(* IEC 61131-3 sources: std_i2980_v2.06_cp053/Source/IMM/ieccontrol/ODC1 (part 11) *)

IF sv_DataState = nReadMoldData THEN
   //loading of mold data in progress
   mbIgnoreProgramSwitchChange := TRUE;
   PrevState := nReadMoldData;
   sv_SequenceDimension.iMaxColumns := 0;
   sv_SequenceDimension.iMaxRows := 0;
ELSIF sv_DataState = nReadSequenceData THEN
   //loading of sequence in progress
   mbIgnoreProgramSwitchChange := TRUE;
   PrevState := nReadSequenceData;
   sv_SequenceDimension.iMaxColumns := 0;
   sv_SequenceDimension.iMaxRows := 0;
END_IF;

IF sv_DataState = nReady AND mbIgnoreProgramSwitchChange THEN

   //loading procedure ready
   mbIgnoreProgramSwitchChange := FALSE;

   //decide if only conditions should be recalculated (after loading sequence)
   //or complete sequence should be created (after program switch changed)
   IF sv_bUseProgramSwitches THEN
      aSetPendingRecalc(RecalcMode := nODCRecalcReloadFiles);
   ELSIF PrevState = nReadMoldData THEN
      aSetPendingRecalc(RecalcMode := nODCRecalcInternal);
   ELSIF PrevState = nReadSequenceData THEN
      aSetPendingRecalc(RecalcMode := nODCRecalcInternal);
   END_IF;

   aDoPendingRecalc();
   IF aDoPendingRecalc.bStartedRecalc THEN
      fbDebugTrace2(nDeviceState, 'recalc because data state change');
   END_IF;

   PrevState := nReady;
END_IF;

@END_Body

@@@BEG_Comment@@@
@TL(0)

@@@END_Comment@@@

@BEG_Body
@TL(34)
(**************************************** WARNING ********************************************
 *** The KEBA Kemro K2 System including software is not intended for safety control tasks! ***
 ***                       For further information see Comment tab!                        ***
 *********************************************************************************************)

IF NOT sv_bODCFilesChanged THEN
   RETURN;
END_IF;

sv_bODCFilesChanged := FALSE;

IF NOT sv_bInitDone THEN
   fbDebugTrace('ignoring sv_bODCFilesChanged because sv_bInitDone is FALSE');
   RETURN;
END_IF;

(* rebuild ODC array immediately with reloading files *)
aSetPendingRecalc(RecalcMode := nODCRecalcReloadFiles);

IF sv_OperationMode >= nHalfAutomatic THEN
   fbDebugTrace('skipping ODC recalc after file change because of OperationMode');
   RETURN;
END_IF;

IF sv_StartedMovements.iStartedMovements > 0 THEN
   fbDebugTrace('skipping ODC recalc after file change because there are started movements');
   RETURN;
END_IF;

aDoPendingRecalc();
IF aDoPendingRecalc.bStartedRecalc THEN
   fbDebugTrace2(nDeviceState, 'recalc because files changed');
END_IF;

@END_Body

@@@BEG_Comment@@@
@TL(1)
React to program switch changes, and recalculate the ODC sequence.
@@@END_Comment@@@

@BEG_Body
@TL(38)
(**************************************** WARNING ********************************************
 *** The KEBA Kemro K2 System including software is not intended for safety control tasks! ***
 ***                       For further information see Comment tab!                        ***
 *********************************************************************************************)

IF sv_iActiveEditors <> 0 THEN
   //teach mode active
   //avoid changing operation mode to HA or FA
   fbLockUnlock.Alarm.AlarmId := erTeachModeActive;
   fbLockUnlock.Mode := nLockAbort;
   fbLockUnlock();

   //reset sv_bUseProgramSwitches immediately after activating teach mode
   //so that "controlled by machine sequencer" is displayed instead of program switches
   sv_bUseProgramSwitches := FALSE;
   RETURN;
ELSE
   fbLockUnlock.Alarm.AlarmId := erTeachModeActive;
   fbLockUnlock.Mode := nUnlock;
   fbLockUnlock();
END_IF;

//teach mode inactive => new sequence programmed by editor
// -> create internal array, calculate safety conditions, do plaus checks
aSetPendingRecalc(RecalcMode := nODCRecalcInternal);

aDoPendingRecalc();
IF aDoPendingRecalc.bStartedRecalc THEN
   fbDebugTrace2(nDeviceState, 'recalc because new sequence from editor');
END_IF;

@END_Body

@@@BEG_Comment@@@
@TL(2)
create internal array and calculate safety conditions after
teachmode becomes inactive
@@@END_Comment@@@

@BEG_Body
@TL(25)
(**************************************** WARNING ********************************************
 *** The KEBA Kemro K2 System including software is not intended for safety control tasks! ***
 ***                       For further information see Comment tab!                        ***
 *********************************************************************************************)

IF sv_iSequenceToRestore = 0 THEN
   RETURN;
END_IF;

IF sv_iSequenceToRestore > cODCSequenceBackupCount THEN
   fbDebugTrace2(nODCInterpreter, 'restoring actual sequence calculated from switches');
   aSetPendingRecalc(RecalcMode := nODCRecalcCylce);
END_IF;

fbDebugTrace2(nODCInterpreter, CONCAT('restoring old sequence ', DINT_TO_STRING(sv_iSequenceToRestore)));
sv_ODCSequence := sv_ODCSequenceBackup[sv_iSequenceToRestore].Sequence;
aSetPendingRecalc(RecalcMode := nODCRecalcSafety);
aDoPendingRecalc(); //FIXME: this may not do more than security recalculation -> otherwise loaded array would be overwritten
IF aDoPendingRecalc.bStartedRecalc THEN
   fbDebugTrace2(nDeviceState, 'recalc because sequence backup is restored');
END_IF;
sv_iSequenceToRestore := 0;
fbDebugTrace2(nODCInterpreter, 'restoring old sequence done');

@END_Body

@@@BEG_Comment@@@
@TL(0)

@@@END_Comment@@@

@BEG_Body
@TL(45)
(**************************************** WARNING ********************************************
 *** The KEBA Kemro K2 System including software is not intended for safety control tasks! ***
 ***                       For further information see Comment tab!                        ***
 *********************************************************************************************)

IF NOT sv_bProgramSwitchChanged THEN
   RETURN;
END_IF;

sv_bProgramSwitchChanged := FALSE;

IF NOT sv_bInitDone THEN
   fbDebugTrace2(nODCInterpreter, 'ignoring program switch change because sv_bInitDone is FALSE');
   RETURN;
END_IF;

IF NOT sv_bUseProgramSwitches THEN
   // ignore changing of program switch if sequence from graphical editor is used
   fbDebugTrace2(nODCInterpreter, 'ignoring program switch change because of sv_bUseProgramSwitches');
   RETURN;
END_IF;

IF mbIgnoreProgramSwitchChange THEN
   fbDebugTrace2(nODCInterpreter, 'ignoring program switch change because of sv_DataState');
   RETURN;
END_IF;

aSetPendingRecalc(RecalcMode := nODCRecalcCylce);

IF sv_OperationMode >= nHalfAutomatic THEN
   fbDebugTrace('skipping ODC recalc after program switch change because of OperationMode');
   RETURN;
END_IF;

IF sv_StartedMovements.iStartedMovements > 0 THEN
   fbDebugTrace('skipping ODC recalc after program switch change because there are started movements');
   RETURN;
END_IF;

(* rebuild ODC array immediately without reloading files *)
aDoPendingRecalc();
IF aDoPendingRecalc.bStartedRecalc THEN
   fbDebugTrace2(nDeviceState, 'recalc because program switch changed');
END_IF;

@END_Body

@@@BEG_Comment@@@
@TL(1)
React to program switch changes, and recalculate the ODC sequence.
@@@END_Comment@@@

@BEG_Body
@TL(39)
(**************************************** WARNING ********************************************
 *** The KEBA Kemro K2 System including software is not intended for safety control tasks! ***
 ***                       For further information see Comment tab!                        ***
 *********************************************************************************************)

IF NOT sv_bActivationChanged THEN
   RETURN;
END_IF;

sv_bActivationChanged := FALSE;

IF NOT sv_bInitDone THEN
   fbDebugTrace('ignoring sv_bActivationChanged because sv_bInitDone is FALSE');
   RETURN;
END_IF;

IF mbIgnoreProgramSwitchChange THEN
   fbDebugTrace2(nODCInterpreter, 'ignoring activation change because of sv_DataState');
   RETURN;
END_IF;

(* recalculate ODC safety without reloading files/recalculating the sequence *)
aSetPendingRecalc(RecalcMode := nODCRecalcSafety);

IF sv_OperationMode >= nHalfAutomatic THEN
   fbDebugTrace('skipping ODC recalc after activation change because of OperationMode');
   RETURN;
END_IF;

IF sv_StartedMovements.iStartedMovements > 0 THEN
   fbDebugTrace('skipping ODC recalc after activation change because there are started movements');
   RETURN;
END_IF;

aDoPendingRecalc();
IF aDoPendingRecalc.bStartedRecalc THEN
   fbDebugTrace2(nDeviceState, 'recalc because activation change');
END_IF;

@END_Body

@@@BEG_Comment@@@
@TL(1)
React to program switch changes, and recalculate the ODC sequence.
@@@END_Comment@@@

@BEG_Body
@TL(8)
(**************************************** WARNING ********************************************
 *** The KEBA Kemro K2 System including software is not intended for safety control tasks! ***
 ***                       For further information see Comment tab!                        ***
 *********************************************************************************************)

b := FCreateODCVersion();
STOP_PROCESS_ALGORITHM();

@END_Body

@@@BEG_Comment@@@
@TL(0)

@@@END_Comment@@@

@BEG_Body
@TL(29)
(**************************************** WARNING ********************************************
 *** The KEBA Kemro K2 System including software is not intended for safety control tasks! ***
 ***                       For further information see Comment tab!                        ***
 *********************************************************************************************)

IF mbIgnoreProgramSwitchChange THEN
   //loading procedure in progress
   RETURN;
END_IF;

IF sv_bUseProgramSwitches THEN
   //activate all devices after a change from
   //machine sequencer mode to program switch mode
   FOR iDevice := 1 TO sv_ODCDeviceMovements.iCount DO
      IF CHECK_REF(sv_ODCDeviceMovements.Devices[iDevice].pbDeviceActivated^) THEN
         sv_ODCDeviceMovements.Devices[iDevice].pbDeviceActivated^ := TRUE;
      END_IF;
   END_FOR;

   //create new sequence depending on the program switches
   //set mode to nODCRecalcReloadFiles because maybe sequence was
   //never created with program switches before
   aSetPendingRecalc(RecalcMode := nODCRecalcReloadFiles);
   aDoPendingRecalc();
   IF aDoPendingRecalc.bStartedRecalc THEN
      fbDebugTrace2(nDeviceState, 'recalc because change to program switch mode');
   END_IF;
END_IF;

@END_Body

@@@BEG_Comment@@@
@TL(1)
trigger creation of sequence by program switches
@@@END_Comment@@@

@BEG_Body
@TL(78)
(**************************************** WARNING ********************************************
 *** The KEBA Kemro K2 System including software is not intended for safety control tasks! ***
 ***                       For further information see Comment tab!                        ***
 *********************************************************************************************)

Pos.iColumn := 1;
Pos.iRow := 1;

DeviceId.CompId := sv_ODCSequence[1,1].iCompId;
DeviceId.IndexId := INT_TO_DINT(sv_ODCSequence[1,1].iIndexId);

//check safety array of first step (ODC.BeginSequence)
bEjectorIgnored := FALSE;
IF mbEjeBwdAtCycleStart THEN
   //ejector must not be bwd when operator switches to HA or FA
   //the ejector bwd movement is done in aRunAutoCylce
   //=> start of cycle should be possible if ejector is not bwd)
   //=> dependency must be modified for this case
   //all other safety relevant movements (mold, cores, ...) must be in the calculated startposition
   EjectorDependency := sv_ODCSequenceInt[1,1].SafetyArray[miIndexEjectorInSafetyArray].Dependency;
   sv_ODCSequenceInt[1,1].SafetyArray[miIndexEjectorInSafetyArray].Dependency := cNoDependency;
   bEjectorIgnored := TRUE;
END_IF;

//check init safety array
//(check all safety relevant devices)
abODCCheckDependencies.aCheck(StepPos := Pos, DeviceIdSelf := DeviceId);
bAllowed := abODCCheckDependencies.aCheck.bAllowed;

//write back the original value
IF bEjectorIgnored THEN
   sv_ODCSequenceInt[1,1].SafetyArray[miIndexEjectorInSafetyArray].Dependency := EjectorDependency;
END_IF;

//check state of not safety relevant devices
//always check even if safety relevant check already failed
SafetyArray := sv_ODCSequenceInt[1,1].SafetyArray;
FOR iDevice := 1 TO sv_ODCDeviceMovements.iCount DO
   DeviceId := sv_ODCDeviceMovements.Devices[iDevice].DeviceId;
   iDefaultMove := sv_ODCDeviceMovements.Devices[iDevice].iDefaultMoveNumber;

   IF (SafetyArray[iDevice].Dependency = cNoDependency) AND (DeviceId.CompId <> cCompODC) THEN
      //device not safety relevant
      IF sv_ODCDeviceMovements.Devices[iDevice].pbDeviceActivated^ AND iDefaultMove <> 0 THEN
         //if device is activated and a default movement is available,
         //the default movement of this device must be in endposition
         fbCheckPosReached(DeviceId := DeviceId,
                           MoveDir := sv_MovementsAvailable[iDefaultMove].pMovementData^.MoveDir,
                           MoveId := sv_MovementsAvailable[iDefaultMove].pMovementData^.MoveId);

         IF NOT fbCheckPosReached.bPosReached THEN
            IF sv_TraceLevel.bODCInterpreter THEN
               fbDebugTrace(CONCAT('cycle start not allowed by default position check of ',
                                   DINT_TO_STRING(DeviceId.CompId), '.', DINT_TO_STRING(DeviceId.IndexId),
                                   ' -> setting alarm ',
                                   GET_ALARM_NAME(fbCheckPosReached.Alarm.AlarmId)));
            END_IF;
            //set according alarm
            SET_ALARM(Name := fbCheckPosReached.Alarm.AlarmId,
                      SubID1 := fbCheckPosReached.Alarm.SubId[1],
                      SubID2 := fbCheckPosReached.Alarm.SubId[2],
                      SubID3 := fbCheckPosReached.Alarm.SubId[3],
                      SubID4 := fbCheckPosReached.Alarm.SubId[4]);
            bAllowed := FALSE;
         END_IF;
      END_IF;
   END_IF;
END_FOR;

IF NOT bAllowed THEN
   IF sv_TraceLevel.bODCInterpreter THEN
      fbDebugTrace('checking cycle start conditions found problems -> switching back to manual mode');
   END_IF;
   //switch away from auto mode if any check fails
   fbAutoManual();
END_IF;

@END_Body

@@@BEG_Comment@@@
@TL(6)
This algorithm checks the start conditions for the cycle if the
operator switches to half or fullauto cycle.
Safety relevant devices must be in the position which they should have according
the programmed cycle.
Not safety relevant devices must be in their default position.
Deactivated devices and devices which have no default position are not checked.
@@@END_Comment@@@

@BEG_Body
@TL(28)
(**************************************** WARNING ********************************************
 *** The KEBA Kemro K2 System including software is not intended for safety control tasks! ***
 ***                       For further information see Comment tab!                        ***
 *********************************************************************************************)

IF sv_TraceLevel.bODCInterpreter THEN
   //trace opmode switch
   IF sv_OperationMode = nSetup THEN
      sOperationMode := 'Setup';
   ELSIF sv_OperationMode = nManual THEN
      sOperationMode := 'Manual';
   ELSIF sv_OperationMode = nHalfAutomatic THEN
      sOperationMode := 'HalfAutomatic';
   ELSIF sv_OperationMode = nFullAutomatic THEN
      sOperationMode := 'FullAutomatic';
   ELSE
      sOperationMode := '???';
   END_IF;
   fbDebugTrace(CONCAT('sv_OperationMode changed to ', sOperationMode));
END_IF;

IF PrevOpMode < nHalfAutomatic AND sv_OperationMode >= nHalfAutomatic THEN
   //check cycle start conditions
   aCheckCycleStartConditions();
END_IF;

PrevOpMode := sv_OperationMode;

@END_Body

@@@BEG_Comment@@@
@TL(0)

@@@END_Comment@@@

@BEG_SfcBody
25 16 17

@BEG_SfcData 2
@StepSeq @RT(4)sseq @F 3
@Step @RT(5)SInit @F @T @F @F @RT(0) @F
@AcbCont @RT(7)unnamed @F 0

@Trans @RT(6)Trans1 @F @T @F @F @T @F @TL(2)
TRUE

@RT(6)Trans1 @F
@Loop @RT(4)loop @F 2
@StepSeq @RT(3)seq @F 5
@Step @RT(5)S_Run @F @F @F @F @RT(0) @F
@AcbCont @RT(7)unnamed @F 2
@Acb @RT(8)Action24 @F @T @RT(1)P @RT(0) @F @F @T @TL(2)
sv_bODCCombinedMoveActive := TRUE;

@F
@Acb @RT(20)ARunCombinedMovement @F @T @RT(1)N @RT(0) @F @F @T @TL(4)
// run a combined movements
abInterpreter.aInterpret();
abInterpreter.aStatus();

@F

@AltBranch @RT(3)alt @F 3
@TransSeq @RT(4)tseq @F 5
@Trans @RT(9)TFinished @F @T @F @F @T @F @TL(2)
abInterpreter.aStatus.bFinished

@RT(6)Trans2 @F
@Step @RT(10)S_Finished @F @F @F @F @RT(0) @F
@AcbCont @RT(7)unnamed @F 1
@Acb @RT(6)ATrace @F @F @RT(1)P @RT(0) @F @F @F @F

@Trans @RT(18)TAllMovementsReady @F @T @F @F @T @F @TL(2)
sv_StartedManualMovements.iStartedMovements = 0

@RT(6)Trans7 @T @TL(2)
Interpreter is finished -> wait untill all movements
are ready  (for example airvalve can still be active)

@Step @RT(17)S_StopInterpreter @F @F @F @F @RT(0) @F
@AcbCont @RT(7)unnamed @F 1
@Acb @RT(16)AStopInterpreter @F @T @RT(1)P @RT(0) @F @F @T @TL(2)
abInterpreter.aStopInterpreterNormal();

@F

@Trans @RT(7)Trans11 @F @T @F @F @T @F @TL(2)
TRUE

@RT(7)Trans11 @F

@TransSeq @RT(4)tseq @F 3
@Trans @RT(10)TNotActive @F @T @F @F @T @F @TL(2)
NOT abInterpreter.aStatus.bActive

@RT(6)Trans5 @F
@Step @RT(11)S_NotActive @F @F @F @F @RT(0) @F
@AcbCont @RT(7)unnamed @F 1
@Acb @RT(15)ATraceNotActive @F @F @RT(1)P @RT(0) @F @F @F @F

@Trans @RT(6)Trans8 @F @T @F @F @T @F @TL(2)
TRUE

@RT(6)Trans8 @F

@TransSeq @RT(4)tseq @F 3
@Trans @RT(6)TError @F @T @F @F @T @F @TL(2)
abInterpreter.aStatus.bError

@RT(6)Trans6 @F
@Step @RT(7)S_Error @F @F @F @F @RT(0) @F
@AcbCont @RT(7)unnamed @F 1
@Acb @RT(11)ATraceError @F @F @RT(1)P @RT(0) @F @F @F @F

@Trans @RT(6)Trans9 @F @T @F @F @T @F @TL(2)
TRUE

@RT(6)Trans9 @F

@Step @RT(8)S_Recalc @F @F @F @F @RT(0) @F
@AcbCont @RT(7)unnamed @F 1
@Acb @RT(16)ADoPendingRecalc @F @F @RT(1)P @RT(0) @F @F @F @F

@Trans @RT(7)Trans12 @F @T @F @F @T @F @TL(2)
TRUE

@RT(7)Trans12 @F
@Step @RT(6)S_Stop @F @F @F @F @RT(0) @F
@AcbCont @RT(7)unnamed @F 1
@Acb @RT(5)AStop @F @T @RT(1)P @RT(0) @F @F @T @TL(3)
sv_bODCCombinedMoveActive := FALSE;
STOP_PROCESS_ALGORITHM();

@F

@Trans @RT(6)Trans4 @F @T @T @T @T @T @TL(2)
TRUE

@RT(6)Trans4 @F

@END_SfcData
@SaActions 4
@SaText @RT(6)ATrace 1 @TL(10)
(**************************************** WARNING ********************************************
 *** The KEBA Kemro K2 System including software is not intended for safety control tasks! ***
 ***                       For further information see Comment tab!                        ***
 *********************************************************************************************)

fbDebugTrace2(nODCInterpreter,'stopping combined movement PA because interpreter has finished');
IF sv_StartedManualMovements.iStartedMovements <> 0 THEN
   fbDebugTrace2(nODCInterpreter,'There were still some movements active at end of a combined movement');
END_IF;

@SaText @RT(11)ATraceError 1 @TL(7)
(**************************************** WARNING ********************************************
 *** The KEBA Kemro K2 System including software is not intended for safety control tasks! ***
 ***                       For further information see Comment tab!                        ***
 *********************************************************************************************)

fbDebugTrace2(nODCInterpreter,'stopping combined movement PA because interpreter reported an error');

@SaText @RT(15)ATraceNotActive 1 @TL(10)
(**************************************** WARNING ********************************************
 *** The KEBA Kemro K2 System including software is not intended for safety control tasks! ***
 ***                       For further information see Comment tab!                        ***
 *********************************************************************************************)

fbDebugTrace2(nODCInterpreter,'stopping combined movement PA because interpreter is not active anymore');
IF sv_StartedManualMovements.iStartedMovements <> 0 THEN
   fbDebugTrace2(nODCInterpreter,'There were still some movements active at end of a combined movement');
END_IF;

@SaText @RT(16)ADoPendingRecalc 1 @TL(14)
(**************************************** WARNING ********************************************
 *** The KEBA Kemro K2 System including software is not intended for safety control tasks! ***
 ***                       For further information see Comment tab!                        ***
 *********************************************************************************************)

IF sv_StartedManualMovements.iStartedMovements = 0 THEN
   //all movements ready
   aDoPendingRecalc();
   IF aDoPendingRecalc.bStartedRecalc THEN
      fbDebugTrace2(nDeviceState, 'recalc because interpreter finished and iStartedMovements = 0');
   END_IF;
END_IF;

@SaTrans 0
@SaExits 0
@END_SfcBody

@@@BEG_Comment@@@
@TL(0)

@@@END_Comment@@@

@BEG_Body
@TL(21)
(**************************************** WARNING ********************************************
 *** The KEBA Kemro K2 System including software is not intended for safety control tasks! ***
 ***                       For further information see Comment tab!                        ***
 *********************************************************************************************)

FOR i := 1 TO sv_StartedManualMovements.iStartedMovements DO

   TmpStepPos := sv_StartedManualMovements.MoveData[i].StepPos;
   IF (TmpStepPos.iColumn <> 0) AND (TmpStepPos.iRow <> 0) THEN
      //if a combined movement (sequence) is active, the supervision of the check conditions
      //is done automatically by the interpreter
      abInterpreter.aCheckConditionsManual(Movement := sv_ODCSequence[TmpStepPos.iColumn][TmpStepPos.iRow], bNoAlarms := FALSE);

      IF NOT abInterpreter.aCheckConditionsManual.bCheckConditionsOk THEN
         //check condition not ok
         abInterpreter.aStopInterpreterError();
      END_IF;
   END_IF;
END_FOR;

@END_Body

@@@BEG_Comment@@@
@TL(4)
supervision of check conditions for single movements in
manual and setup mode
For combined movements and in half and fullauto cycle the supervision
is done by the interpreter
@@@END_Comment@@@

@BEG_Body
@TL(23)
(**************************************** WARNING ********************************************
 *** The KEBA Kemro K2 System including software is not intended for safety control tasks! ***
 ***                       For further information see Comment tab!                        ***
 *********************************************************************************************)

//Cycle time - from start to start
IF mbCycleTimeRunning THEN

   IF mbResetCycleTime THEN
      fbTonCycleTime(IN := FALSE);
      mbResetCycleTime := FALSE;
   END_IF;

   fbTonCycleTime(IN := TRUE,
                  PT := t#20d);

   b := WRITE_SV_DIRECT(sv_dCycleTime, fbTonCycleTime.ET);

   IF sv_dCycleTime > sv_dMaxCycleTime THEN
      SET_ALARM(Name := erCycleTimeExceeded);
   END_IF;
END_IF;

@END_Body

@@@BEG_Comment@@@
@TL(0)

@@@END_Comment@@@

@BEG_Body
@TL(19)
(**************************************** WARNING ********************************************
 *** The KEBA Kemro K2 System including software is not intended for safety control tasks! ***
 ***                       For further information see Comment tab!                        ***
 *********************************************************************************************)

//Cycle time machine - from start to end of cycle
IF mbCycleTimeRunning AND mbCycleTimeMachineRunning THEN

   IF mbResetCycleTimeMachine THEN
      fbTonCycleTimeMachine(IN := FALSE);
      mbResetCycleTimeMachine := FALSE;
   END_IF;

   fbTonCycleTimeMachine(IN := TRUE,
                         PT := t#20d);

   b := WRITE_SV_DIRECT(sv_dCycleTimeMachine, fbTonCycleTimeMachine.ET);
END_IF;

@END_Body

@@@BEG_Comment@@@
@TL(0)

@@@END_Comment@@@

@BEG_Body
@TL(22)
(**************************************** WARNING ********************************************
 *** The KEBA Kemro K2 System including software is not intended for safety control tasks! ***
 ***                       For further information see Comment tab!                        ***
 *********************************************************************************************)

IF sv_bSequenceInterruption THEN
   IF sv_TraceLevel.bODCInterpreter THEN
      dummy := Print('***** INTERRUPT SEQUENCE *****');
   END_IF;
   mbStopAfterCycle := TRUE;
   abInterpreter.aInterruptSequence();
ELSE
   sv_bStepBwdActive := FALSE;
   IF sv_OperationMode >= nHalfAutomatic THEN
      IF sv_TraceLevel.bODCInterpreter THEN
         dummy := Print('***** CONTINUE SEQUENCE *****');
      END_IF;
      abInterpreter.aContinueSequence();
      mbStopAfterCycle := FALSE;
   END_IF;
END_IF;

@END_Body

@@@BEG_Comment@@@
@TL(0)

@@@END_Comment@@@

@BEG_Body
@TL(40)
(**************************************** WARNING ********************************************
 *** The KEBA Kemro K2 System including software is not intended for safety control tasks! ***
 ***                       For further information see Comment tab!                        ***
 *********************************************************************************************)

//get inverse movement
iMoveIdInverse := sv_MovementsAvailable[iMoveNr].pMovementData^.iMoveIdInverseMovement;
IF iMoveIdInverse = cMinMoveIdent THEN
   //no inverse movement defined
   //set alarm if moenet does not belong to ODC - function unit
   IF (sv_MovementsAvailable[iMoveNr].DeviceId <> sv_DeviceId) THEN
      SET_ALARM(Name := erNoInverseMovement,
                SubID1 := sv_MovementsAvailable[iMoveNr].DeviceId.CompId,
                SubID2 := sv_MovementsAvailable[iMoveNr].DeviceId.IndexId,
                SubID3 := sv_MovementsAvailable[iMoveNr].pMovementData^.MoveId);
   END_IF;

   RETURN; //return here
END_IF;

iFuIndex := sv_MovementsAvailable[iMoveNr].iFuIndex;
FOR i := 1 TO sv_ODCDeviceMovements.Devices[iFuIndex].iNumberOfMovements DO
   IF sv_ODCDeviceMovements.Devices[iFuIndex].Movements[i]^.MoveId = iMoveIdInverse THEN
      //inverse movement found => try to start it
      aStartSingleMovement(DeviceId := sv_ODCDeviceMovements.Devices[iFuIndex].DeviceId,
                           MoveDir := sv_ODCDeviceMovements.Devices[iFuIndex].Movements[i]^.MoveDir,
                           MoveId := sv_ODCDeviceMovements.Devices[iFuIndex].Movements[i]^.MoveId,
                           IntermediateCond := 0,
                           bNeedCheckSafety := (sv_ODCDeviceMovements.Devices[iFuIndex].Movements[i]^.iSafetyIdentifier > 0));

      IF aStartSingleMovement.bStarted THEN
         mActiveStepBwdMovements[iColumn].DeviceId := sv_ODCDeviceMovements.Devices[iFuIndex].DeviceId;
         mActiveStepBwdMovements[iColumn].MoveId := sv_ODCDeviceMovements.Devices[iFuIndex].Movements[i]^.MoveId;
         mActiveStepBwdMovements[iColumn].MoveDir := sv_ODCDeviceMovements.Devices[iFuIndex].Movements[i]^.MoveDir;
      END_IF;

      EXIT;
   END_IF;
END_FOR;

@END_Body

@@@BEG_Comment@@@
@TL(0)

@@@END_Comment@@@

@BEG_Body
@TL(21)
(**************************************** WARNING ********************************************
 *** The KEBA Kemro K2 System including software is not intended for safety control tasks! ***
 ***                       For further information see Comment tab!                        ***
 *********************************************************************************************)

IF NOT sv_bSequenceInterruption THEN
   //button is only working if sequence is interrupted
   RETURN;
END_IF;

IF di_StepFwd THEN
   //trigger interpreter to execute the next step(s)
   IF sv_StartedManualMovements.iStartedMovements = 0 THEN
      //ignore step fwd button if any movment is active
      abInterpreter.aEnableNextStep();
   END_IF;
ELSE
   //stop actually executed step(s)
   abInterpreter.aInterruptSequence();
END_IF;

@END_Body

@@@BEG_Comment@@@
@TL(0)

@@@END_Comment@@@

@BEG_Body
@TL(51)
(**************************************** WARNING ********************************************
 *** The KEBA Kemro K2 System including software is not intended for safety control tasks! ***
 ***                       For further information see Comment tab!                        ***
 *********************************************************************************************)

IF NOT sv_bSequenceInterruption THEN
   //button is only working if sequence is interrupted
   RETURN;
END_IF;

IF di_StepBwd THEN

   IF sv_StartedManualMovements.iStartedMovements <> 0 THEN
      //ignore step bwd button if any movement is still active
      RETURN;
   END_IF;

   sv_bStepBwdActive := TRUE;

   //get actual active lines and find the inverse movements
   FOR iColumn := 1 TO sv_iUsedColumns DO
      IF sv_InterpreterParallelInfo[iColumn].bColumnActive THEN
         //it is possible that the sequence was interrupted during waiting
         //for completion of a parallel tree -> in this case the line number must be decreased
         IF (sv_ODCSequence[iColumn, sv_InterpreterParallelInfo[iColumn].iRow].iMoveId = cMoveEndParallel) THEN
            abInterpreter.aDecreaseRow(bStartInActualLine := FALSE,
                                       iColumn := iColumn,
                                       iEndRow := 1);
         ELSIF (sv_ODCSequence[iColumn, sv_InterpreterParallelInfo[iColumn].iRow].iMoveId = cMoveStartParallel) OR
            (sv_ODCSequence[iColumn, sv_InterpreterParallelInfo[iColumn].iRow].iMoveId = cMoveStartParallelOpen) THEN
            //stepping bwd stopped during waiting for parallel trees
            //-> check actual state of this tree
            abInterpreter.aDecreaseRow(bStartInActualLine := TRUE,
                                       iColumn := iColumn,
                                       iEndRow := 1);
         END_IF;

         iActiveMoveNr := sv_ODCSequenceInt[iColumn, sv_InterpreterParallelInfo[iColumn].iRow].iMoveNumber;
         IF iActiveMoveNr > cMoveNone THEN
            aStartInverseMovement(iMoveNr := iActiveMoveNr,
                                 iColumn := iColumn);
         END_IF;
      END_IF;
   END_FOR;
ELSE
   //stop actually executed step(s)
   abInterpreter.aInterruptSequence();

   sv_bStepBwdActive := FALSE;
END_IF;

@END_Body

@@@BEG_Comment@@@
@TL(0)

@@@END_Comment@@@

@BEG_Body
@TL(51)
(**************************************** WARNING ********************************************
 *** The KEBA Kemro K2 System including software is not intended for safety control tasks! ***
 ***                       For further information see Comment tab!                        ***
 *********************************************************************************************)

IF sv_iInitOK <> 20 THEN
   dummy := Print('!!! evModifyCycleStartCondition event ignored !!!');
   RETURN; //ignore event because machine sequence is not created
END_IF;

//save event data
eventData := evModifyCycleStartCondData;

//get index of this device in the safety array
iFuIndex := 0;
FOR i := 1 TO sv_ODCDeviceMovements.iCount DO
   IF sv_ODCDeviceMovements.Devices[i].DeviceId = eventData.DeviceId THEN
      iFuIndex := i;
      EXIT;
   END_IF;
END_FOR;

IF iFuIndex = 0 THEN
   RETURN; //device not found
END_IF;

IF (eventData.iMode = 1) THEN
   //get movement number
   fbGetMoveNumber(DeviceId := eventData.DeviceId,
                  MoveId := eventData.MoveId,
                  MoveDir := eventData.MoveDir);

   IF fbGetMoveNumber.bFound THEN
      iMoveNr := fbGetMoveNumber.iMoveNumber;
   ELSE
      RETURN; //movement not found
   END_IF;

   //add this movement as additional start condition of this device
   fbAddDependency(iFuIndex := iFuIndex,
                   iMoveNr := iMoveNr,
                   iCount := eventData.iCount,
                   iMode := 1,
                   Dependency := sv_ODCSequenceInt[1,1].SafetyArray);

ELSE
   ; //unsupported mode
END_IF;

@END_Body

@@@BEG_Comment@@@
@TL(0)

@@@END_Comment@@@
@END_Body

@END_Contents
@@@BEG_Password@@@
NGhzZm9kYzQ=
@@@END_Password@@@

(* ---- ABODCCheckDependencies.pu ---- *)
(*
Called by aCheck
*)

IMPORT_OVER_LISTFILE
 SET_ALARM
, CHECK_REF
, cCompCore
, cCompMold
, cMaxDeviceMovements
, cMaxIntermediateConditions
, cFirstBit
, tsGlbSafetyData
, tyMovementRegisterList
, tyODCSequenceInternal
, tsODCDeviceMovementList
, ABSEInterpreter
, tsSafetyHMICom
, tsODCStepPos
, tsDeviceId
, tsAlarm
, FBSetStepState

END_IMPORT

ALGORITHM_BLOCK ABODCCheckDependencies #DUMMY_EDIT_BLOCK

SYSTEM_VAR
 sv_MovementsAvailable : tyMovementRegisterList;
 sv_ODCSequenceInt : tyODCSequenceInternal;
 sv_ODCDeviceMovements : tsODCDeviceMovementList (* list of all devices that registered movements for the ODC *);
 sv_bOverrideCoreSafety : BOOL (* overrides safety settings for core movements in setup mode *);
 sv_bOverrideEjectorSafety : BOOL (* overrides safety settings for ejector movements in setup mode *);
END_VAR

SYSTEM_VAR_IN
 sv_SafetyHMICom : tsSafetyHMICom;
END_VAR

SYSTEM_OBJECT
 erODCComponentLocked : ALARM;
 TaskVis : TASK;
 erCompNotInCorrectPosition : ALARM;
END_OBJECT

VAR_EXTERNAL
 g_SafetyData : tsGlbSafetyData;
 g_iODCMoveDevicesRegistered : DINT;
END_VAR

VAR
 abSEInterpreter : ABSEInterpreter;
 mbOverrideDefaultSafety : BOOL;
END_VAR

ALGORITHM aCheckInstances

VAR_INPUT
 Dependency : LWORD;
 iDeviceIndex : DINT;
 iMoveInDevice : DINT;
END_VAR

VAR_OUTPUT
 bAllowed : BOOL;
END_VAR

VAR_TEMP
 i : DINT;
 k : DINT;
END_VAR

VAR
 tmpDependency : LWORD;
 iBegin : DINT;
 iInstanceableMovement : DINT;
END_VAR
#BEGIN_EDIT_BLOCK
(**************************************** WARNING ********************************************
 *** The KEBA Kemro K2 System including software is not intended for safety control tasks! ***
 ***                       For further information see Comment tab!                        ***
 *********************************************************************************************)

bAllowed := FALSE;

//find out if it is the first, second, third or fourth instanceable movement in this function unit
iInstanceableMovement := 1;
FOR k := 1 TO cMaxSRInstanceableMovements DO
   IF iMoveInDevice = sv_ODCDeviceMovements.Devices[iDeviceIndex].InstanceableMovements[k] THEN
      iInstanceableMovement := k;
      EXIT;
   END_IF;
END_FOR;

iBegin := cMaxDeviceMovements + ((iInstanceableMovement - 1) * cMaxIntermediateConditions);
tmpDependency := SHL(Dependency, iBegin);

FOR i := 1 TO cMaxIntermediateConditions DO

   tmpDependency := tmpDependency AND cFirstBit;
   IF tmpDependency = cFirstBit THEN
      //bit set => check PosReached of this instance
      bAllowed := sv_ODCDeviceMovements.Devices[iDeviceIndex].Movements[iMoveInDevice]^.InstanceData.pPosReachedArray^[i];

      IF bAllowed THEN
         //movement with posReached = TRUE found -> exit
         EXIT;
      END_IF;
   END_IF;

   tmpDependency := SHL(Dependency, (iBegin + i));

END_FOR;

;#END_EDIT_BLOCK END_ALGORITHM

(*
check safety array for the given step
*)

ALGORITHM aCheckInternal

VAR_INPUT
 StepPos : tsODCStepPos;
 DeviceIdSelf : tsDeviceId;
 bNoAlarmsAndStepState : BOOL (* TRUE: only check dependencies and do not set alarms and stepstate *);
END_VAR

VAR_OUTPUT
 bAllowed : BOOL;
 iNotOkCount : DINT;
END_VAR

VAR_TEMP
 iDevice : DINT;
 iMoveInDevice : DINT;
 i : DINT (* movement number at the given StepPos *);
END_VAR

VAR
 tmpDependency : LWORD;
 Alarm : tsAlarm;
 Dependency : LWORD;
 bTmp : BOOL;
 fbSetStepState : FBSetStepState;
 dummy : DINT;
 bTraced : BOOL;
 iSafetyIdentifier : DINT;
 DeviceId : tsDeviceId;
 bOverrideSafety : BOOL;
 bDeviceOk : BOOL;
 iValidMovements : DINT;
END_VAR
#BEGIN_EDIT_BLOCK
(**************************************** WARNING ********************************************
 *** The KEBA Kemro K2 System including software is not intended for safety control tasks! ***
 ***                       For further information see Comment tab!                        ***
 *********************************************************************************************)

//check safety array for one step
iNotOkCount := 0;
bAllowed := TRUE;

// when iColumn or iRow = 0 then the movement ist not
// present in the auto cycle (and not safety relevant)
IF StepPos.iColumn = 0 OR StepPos.iRow = 0 THEN
   RETURN;
END_IF;

i := sv_ODCSequenceInt[StepPos.iColumn][StepPos.iRow].iMoveNumber;
IF i = 0 THEN
   //avoid out of range errors
   IF NOT bTraced THEN
      //only trace once and not cyclically
      dummy := Print('!! ABODCCheckDependencies: can not check conditions for movement with move nr. = 0 !!');
      dummy := Print('!! DeviceId: %d/%d  column: %d row: %d !!',DeviceIdSelf.CompId, DeviceIdSelf.IndexId, StepPos.iColumn, StepPos.iRow);
      bTraced := TRUE;
   END_IF;

   bAllowed := FALSE;
   RETURN;
ELSE
   bTraced := FALSE;
END_IF;

iSafetyIdentifier := sv_MovementsAvailable[i].pMovementData^.iSafetyIdentifier;

IF ((NOT mbOverrideDefaultSafety) OR (iSafetyIdentifier = 3)) THEN

   FOR iDevice := 1 TO g_iODCMoveDevicesRegistered DO

      //check override flags
      bOverrideSafety := FALSE;
      DeviceId := sv_ODCDeviceMovements.Devices[iDevice].DeviceId;
      IF ((NOT g_SafetyData.bAvailable) AND sv_bOverrideCoreSafety) AND // override core safety only available if no safetyeditor
         DeviceIdSelf.CompId = cCompCore AND
         (DeviceId.CompId = cCompCore OR DeviceId.CompId = cCompMold OR DeviceId.CompId = cCompEjector) THEN
         (* allow core movements even if mold, other cores or ejector are not in correct position *)
         bOverrideSafety := TRUE;
      END_IF;

      IF ((NOT g_SafetyData.bAvailable) AND sv_bOverrideEjectorSafety) AND // override ejector safety only available if no safetyeditor
         DeviceIdSelf.CompId = cCompEjector AND
         (DeviceId.CompId = cCompCore OR DeviceId.CompId = cCompMold OR DeviceId.CompId = cCompEjector) THEN
         (* allow ejector movements even if mold, cores or possibly other ejectors are not in correct position *)
         bOverrideSafety := TRUE;
      END_IF;

      //check all devices in the safety array
      Dependency := sv_ODCSequenceInt[StepPos.iColumn,StepPos.iRow].SafetyArray[iDevice].Dependency;
      IF (Dependency = cNoDependency) OR bOverrideSafety THEN
         //device is not safety relevant or override is activated
         bDeviceOk := TRUE;
      ELSE
         tmpDependency := Dependency;
         bDeviceOk := FALSE;
         iValidMovements := 0;
         FOR iMoveInDevice := 1 TO sv_ODCDeviceMovements.Devices[iDevice].iNumberOfMovements DO
            //check every movement in this device
            tmpDependency := tmpDependency AND cFirstBit;
            IF tmpDependency = cFirstBit THEN

               iValidMovements := iValidMovements + 1;

               //bit set => check posReached of this movement
               IF sv_ODCDeviceMovements.Devices[iDevice].Movements[iMoveInDevice]^.bInstanceable THEN
                  //instanceable movement => check instances
                  aCheckInstances(Dependency := Dependency,
                                 iDeviceIndex := iDevice,
                                 iMoveInDevice := iMoveInDevice);
                  bTmp := aCheckInstances.bAllowed;
               ELSE
                  bTmp := CHECK_REF(sv_ODCDeviceMovements.Devices[iDevice].Movements[iMoveInDevice]^.pbPosReached^) AND
                              sv_ODCDeviceMovements.Devices[iDevice].Movements[iMoveInDevice]^.pbPosReached^;
               END_IF;

               IF bTmp THEN
                  //valid movement with posReached = TRUE in this device found
                  bDeviceOk := TRUE;
                  EXIT;
               ELSE
                  //continue checking this device and save alarm temporary
                  Alarm := sv_ODCDeviceMovements.Devices[iDevice].Movements[iMoveInDevice]^.Alarm;
               END_IF;
            END_IF;
            tmpDependency := SHL(Dependency, iMoveInDevice);

         END_FOR; //end_for checking all movements in one device

         IF NOT bDeviceOk THEN
            //set correct alarm
            IF NOT bNoAlarmsAndStepState THEN
               IF iValidMovements > 1 THEN
                  //two or more allowed movements: set common alarm erCompNotInCorrectPosition
                  SET_ALARM(Name := erCompNotInCorrectPosition,
                           SubID1 := sv_ODCDeviceMovements.Devices[iDevice].DeviceId.CompId,
                           SubID2 := sv_ODCDeviceMovements.Devices[iDevice].DeviceId.IndexId);
               ELSE
                  //only one valid movement: set alarm of this movement
                  IF (Alarm.AlarmId <> EMPTY) THEN
                     SET_ALARM(Name := Alarm.AlarmId,
                           SubID1 := Alarm.SubId[1],
                           SubID2 := Alarm.SubId[2],
                           SubID3 := Alarm.SubId[3],
                           SubID4 := Alarm.SubId[4],
                           Param1 := Alarm.Param1,
                           Param2 := Alarm.Param2);
                  ELSE
                     SET_ALARM(Name   := erODCComponentLocked,
                                 SubID1 := DeviceIdSelf.CompId,
                                 SubID2 := DeviceIdSelf.IndexId,
                                 SubID3 := sv_ODCDeviceMovements.Devices[iDevice].DeviceId.CompId,
                                 SubID4 := sv_ODCDeviceMovements.Devices[iDevice].DeviceId.IndexId);
                  END_IF;
               END_IF; //end_if iValidMovements
            END_IF;  //end_if bNoAlarmsAndStepState

            //increase counter of not fulfilled conditions
            iNotOkCount := iNotOkCount + 1;

         END_IF; //end_if NOT bDeviceOk

      END_IF; //end_if no dependency or override
      bAllowed := bAllowed AND bDeviceOk;
   END_FOR;  //end_for of checking all devices
END_IF;

IF (iSafetyIdentifier = 1) THEN
   bAllowed := bAllowed AND abSEInterpreter.fCheckMovement(StepPos);
END_IF;

IF (NOT bAllowed) AND (NOT bNoAlarmsAndStepState) THEN
   fbSetStepState(StepPos := StepPos, StepState := nStateError);
END_IF;

;#END_EDIT_BLOCK END_ALGORITHM

(*
Check the dependencies of a ODC movement.
Iterates over the dependency array of the step selected by StepPos
and checks the pos reached flags on those movement.
If StepPos.iColumn or StepPos.iRow is 0 then the movement is always allowed.
*)

ALGORITHM aCheck

VAR_INPUT
 StepPos : tsODCStepPos (* Step for which dependencies are checked *);
 DeviceIdSelf : tsDeviceId (* DeviceId used for error message *);
 bNoAlarmsAndStepState : BOOL (* TRUE: only check dependencies and do not set alarms and stepstate *);
END_VAR

VAR_OUTPUT
 bAllowed : BOOL (* Dependencies are fulfilled *);
 iNotOkCount : DINT (* number of conditions which are not ok *);
END_VAR
#BEGIN_EDIT_BLOCK
(**************************************** WARNING ********************************************
 *** The KEBA Kemro K2 System including software is not intended for safety control tasks! ***
 ***                       For further information see Comment tab!                        ***
 *********************************************************************************************)

aCheckInternal(StepPos := StepPos, DeviceIdSelf := DeviceIdSelf, bNoAlarmsAndStepState := bNoAlarmsAndStepState);
bAllowed := aCheckInternal.bAllowed;
iNotOkCount := aCheckInternal.iNotOkCount;

;#END_EDIT_BLOCK END_ALGORITHM

POSTUPDATE_ALGORITHM pOverrideDefaultSafety ON TaskVis WITH sv_SafetyHMICom.bOverrideDefaultSafety

#BEGIN_EDIT_BLOCK
mbOverrideDefaultSafety := sv_SafetyHMICom.bOverrideDefaultSafety;

;#END_EDIT_BLOCK END_ALGORITHM

END_ALGORITHM_BLOCK

#END_OF_IEC_PART

@Puma @IecEditor 6 96 @Pou 25
@@@BEG_Comment@@@
Called by aCheck
@@@END_Comment@@@

@BEG_Contents

@BEG_Func
@RT(17)FuncTreeContainer
2
@Var @RT(9)SET_ALARM @RT(0) @T @T @DERIVED 0 @F @RT(23)KEBA_STANDARD_PROCEDURE @F
@T
@BEG_Attrib
0 @RT(0) @RT(0)
@END_Attrib
1 1 @F @F @F @F

@Var @RT(9)CHECK_REF @RT(0) @T @T @DERIVED 0 @F @RT(23)KEBA_STANDARD_PROCEDURE @F
@T
@BEG_Attrib
0 @RT(0) @RT(0)
@END_Attrib
1 1 @F @F @F @F

@END_Func

@BEG_Const
@RT(18)ConstTreeContainer
5
@Var @RT(9)cCompCore @RT(0) @T @F @DT @RT(4)DINT @RT(0) @T @T @BASIC 0 @F
@F @F
@T
@BEG_Attrib
0 @RT(3)109 @RT(14)Component Core
@END_Attrib
1 1 @F @F @F @F

@Var @RT(9)cCompMold @RT(0) @T @F @DT @RT(4)DINT @RT(0) @T @T @BASIC 0 @F
@F @F
@T
@BEG_Attrib
0 @RT(3)101 @RT(14)Component Mold
@END_Attrib
1 1 @F @F @F @F

@Var @RT(19)cMaxDeviceMovements @RT(0) @T @F @DT @RT(4)DINT @RT(0) @T @T @BASIC 0 @F
@F @F
@T
@BEG_Attrib
0 @RT(2)20 @RT(34)max number of movements per device
@END_Attrib
1 1 @F @F @F @F

@Var @RT(26)cMaxIntermediateConditions @RT(0) @T @F @DT @RT(4)DINT @RT(0) @T @T @BASIC 0 @F
@F @F
@T
@BEG_Attrib
0 @RT(2)10 @RT(38)max. number of intermediate conditions
@END_Attrib
1 1 @F @F @F @F

@Var @RT(9)cFirstBit @RT(0) @T @F @DT @RT(5)LWORD @RT(0) @T @T @BASIC 0 @F
@F @F
@T
@BEG_Attrib
0 @RT(19)16#8000000000000000 @RT(0)
@END_Attrib
1 1 @F @F @F @F

@END_Const

@BEG_Export

@BEG_Kind
@ALGORITHM_BLOCK @RT(22)ABODCCheckDependencies @STRUCTURED_TEXT
@RT(0) @RT(0) @RT(0)
@END_Kind

@BEG_Dcl
@RT(16)DclTreeContainer
13
@Var @RT(12)g_SafetyData @RT(0) @T @T @DERIVED 0 @T @T @DT @RT(15)tsGlbSafetyData @RT(0) @T @T @UNKNOWN 0 @F
@F @F
@T
@BEG_Attrib
3 @RT(0) @RT(0) @RT(0)
@END_Attrib
1 6 @F @F @F @F

@Var @RT(21)sv_MovementsAvailable @RT(0) @T @T @DERIVED 0 @T @T @DT @RT(22)tyMovementRegisterList @RT(0) @T @T @UNKNOWN 0 @F
@F @F
@T
@BEG_Attrib
3 @RT(0) @RT(0) @RT(0)
@END_Attrib
1 8 @F @F @F @F

@Var @RT(17)sv_ODCSequenceInt @RT(0) @T @T @DERIVED 0 @T @T @DT @RT(21)tyODCSequenceInternal @RT(0) @T @T @UNKNOWN 0 @F
@F @F
@T
@BEG_Attrib
3 @RT(0) @RT(0) @RT(0)
@END_Attrib
1 8 @F @F @F @F

@Var @RT(21)sv_ODCDeviceMovements @RT(0) @T @T @DERIVED 0 @T @T @DT @RT(23)tsODCDeviceMovementList @RT(0) @T @T @UNKNOWN 0 @F
@F @F
@T
@BEG_Attrib
3 @RT(0) @RT(57)list of all devices that registered movements for the ODC @RT(0)
@END_Attrib
1 8 @F @F @F @F

@Var @RT(20)erODCComponentLocked @RT(0) @T @T @RENAMED 0 @T @T @DT @RT(5)ALARM @RT(0) @T @T @BASIC 0 @F
@F @F
@T
@BEG_Attrib
3 @RT(0) @RT(0) @RT(0)
@END_Attrib
1 7 @F @F @F @F

@Var @RT(15)abSEInterpreter @RT(0) @T @T @DERIVED 0 @T @T @DT @RT(15)ABSEInterpreter @RT(0) @T @T @UNKNOWN 0 @F
@F @F
@T
@BEG_Attrib
3 @RT(0) @RT(0) @RT(0)
@END_Attrib
1 0 @F @F @F @F

@Var @RT(15)sv_SafetyHMICom @RT(0) @T @T @DERIVED 0 @T @T @DT @RT(14)tsSafetyHMICom @RT(0) @T @T @UNKNOWN 0 @F
@F @F
@T
@BEG_Attrib
3 @RT(0) @RT(0) @RT(0)
@END_Attrib
1 9 @F @F @F @F

@Var @RT(22)sv_bOverrideCoreSafety @RT(0) @T @T @RENAMED 0 @T @T @DT @RT(4)BOOL @RT(0) @T @T @BASIC 0 @F
@F @F
@T
@BEG_Attrib
3 @RT(0) @RT(58)overrides safety settings for core movements in setup mode @RT(0)
@END_Attrib
1 8 @F @F @F @F

@Var @RT(25)sv_bOverrideEjectorSafety @RT(0) @T @F @DT @RT(4)BOOL @RT(0) @T @T @BASIC 0 @F
@F @F
@T
@BEG_Attrib
3 @RT(0) @RT(61)overrides safety settings for ejector movements in setup mode @RT(0)
@END_Attrib
1 8 @F @F @F @F

@Var @RT(7)TaskVis @RT(0) @T @T @RENAMED 0 @T @T @DT @RT(4)TASK @RT(0) @T @T @BASIC 0 @F
@F @F
@T
@BEG_Attrib
3 @RT(0) @RT(0) @RT(0)
@END_Attrib
1 7 @F @F @F @F

@Var @RT(23)mbOverrideDefaultSafety @RT(0) @T @F @DT @RT(4)BOOL @RT(0) @T @T @BASIC 0 @F
@F @F
@T
@BEG_Attrib
3 @RT(0) @RT(0) @RT(0)
@END_Attrib
1 0 @F @F @F @F

@Var @RT(27)g_iODCMoveDevicesRegistered @RT(0) @T @F @DT @RT(4)DINT @RT(0) @T @T @BASIC 0 @F
@F @F
@T
@BEG_Attrib
3 @RT(0) @RT(0) @RT(0)
@END_Attrib
1 6 @F @F @F @F

@Var @RT(26)erCompNotInCorrectPosition @RT(0) @T @F @DT @RT(5)ALARM @RT(0) @T @T @BASIC 0 @F
@F @F
@T
@BEG_Attrib
3 @RT(0) @RT(0) @RT(0)
@END_Attrib
1 7 @F @F @F @F

@END_Dcl

@END_Export

@BEG_Body

4

@BEG_Export

@BEG_Algo
@ALGORITHM @RT(15)aCheckInstances @STRUCTURED_TEXT
@RT(0) @RT(0) @RT(0) @F @F
@END_Algo

@BEG_Dcl
@RT(16)DclTreeContainer
9
@Var @RT(10)Dependency @RT(0) @T @F @DT @RT(5)LWORD @RT(0) @T @T @BASIC 0 @F
@F @F
@T
@BEG_Attrib
3 @RT(0) @RT(0) @RT(0)
@END_Attrib
1 1 @F @F @F @F

@Var @RT(12)iDeviceIndex @RT(0) @T @F @DT @RT(4)DINT @RT(0) @T @T @BASIC 0 @F
@F @F
@T
@BEG_Attrib
3 @RT(0) @RT(0) @RT(0)
@END_Attrib
1 1 @F @F @F @F

@Var @RT(13)iMoveInDevice @RT(0) @T @F @DT @RT(4)DINT @RT(0) @T @T @BASIC 0 @F
@F @F
@T
@BEG_Attrib
3 @RT(0) @RT(0) @RT(0)
@END_Attrib
1 1 @F @F @F @F

@Var @RT(8)bAllowed @RT(0) @T @F @DT @RT(4)BOOL @RT(0) @T @T @BASIC 0 @F
@F @F
@T
@BEG_Attrib
3 @RT(0) @RT(0) @RT(0)
@END_Attrib
1 3 @F @F @F @F

@Var @RT(13)tmpDependency @RT(0) @T @F @DT @RT(5)LWORD @RT(0) @T @T @BASIC 0 @F
@F @F
@T
@BEG_Attrib
3 @RT(0) @RT(0) @RT(0)
@END_Attrib
1 0 @F @F @F @F

@Var @RT(6)iBegin @RT(0) @T @F @DT @RT(4)DINT @RT(0) @T @T @BASIC 0 @F
@F @F
@T
@BEG_Attrib
3 @RT(0) @RT(0) @RT(0)
@END_Attrib
1 0 @F @F @F @F

@Var @RT(1)i @RT(0) @T @F @DT @RT(4)DINT @RT(0) @T @T @BASIC 0 @F
@F @F
@T
@BEG_Attrib
3 @RT(0) @RT(0) @RT(0)
@END_Attrib
1 4 @F @F @F @F

@Var @RT(21)iInstanceableMovement @RT(0) @T @F @DT @RT(4)DINT @RT(0) @T @T @BASIC 0 @F
@F @F
@T
@BEG_Attrib
3 @RT(0) @RT(0) @RT(0)
@END_Attrib
1 0 @F @F @F @F

@Var @RT(1)k @RT(0) @T @F @DT @RT(4)DINT @RT(0) @T @T @BASIC 0 @F
@F @F
@T
@BEG_Attrib
3 @RT(0) @RT(0) @RT(0)
@END_Attrib
1 4 @F @F @F @F

@END_Dcl

@END_Export

@BEG_Export

@BEG_Algo
@ALGORITHM @RT(14)aCheckInternal @STRUCTURED_TEXT
@RT(0) @RT(0) @RT(0) @F @F
@END_Algo

@BEG_Dcl
@RT(16)DclTreeContainer
20
@Var @RT(7)StepPos @RT(0) @T @T @DERIVED 0 @T @T @DT @RT(12)tsODCStepPos @RT(0) @T @T @UNKNOWN 0 @F
@F @F
@T
@BEG_Attrib
3 @RT(0) @RT(0) @RT(0)
@END_Attrib
1 1 @F @F @F @F

@Var @RT(12)DeviceIdSelf @RT(0) @T @T @DERIVED 0 @T @T @DT @RT(10)tsDeviceId @RT(0) @T @T @UNKNOWN 0 @F
@F @F
@T
@BEG_Attrib
3 @RT(0) @RT(0) @RT(0)
@END_Attrib
1 1 @F @F @F @F

@Var @RT(21)bNoAlarmsAndStepState @RT(0) @T @F @DT @RT(4)BOOL @RT(0) @T @T @BASIC 0 @F
@F @F
@T
@BEG_Attrib
3 @RT(0) @RT(65)TRUE: only check dependencies and do not set alarms and stepstate @RT(0)
@END_Attrib
1 1 @F @F @F @F

@Var @RT(8)bAllowed @RT(0) @T @F @DT @RT(4)BOOL @RT(0) @T @T @BASIC 0 @F
@F @F
@T
@BEG_Attrib
3 @RT(0) @RT(0) @RT(0)
@END_Attrib
1 3 @F @F @F @F

@Var @RT(13)tmpDependency @RT(0) @T @F @DT @RT(5)LWORD @RT(0) @T @T @BASIC 0 @F
@F @F
@T
@BEG_Attrib
3 @RT(0) @RT(0) @RT(0)
@END_Attrib
1 0 @F @F @F @F

@Var @RT(5)Alarm @RT(0) @T @T @DERIVED 0 @T @T @DT @RT(7)tsAlarm @RT(0) @T @T @UNKNOWN 0 @F
@F @F
@T
@BEG_Attrib
3 @RT(0) @RT(0) @RT(0)
@END_Attrib
1 0 @F @F @F @F

@Var @RT(10)Dependency @RT(0) @T @F @DT @RT(5)LWORD @RT(0) @T @T @BASIC 0 @F
@F @F
@T
@BEG_Attrib
3 @RT(0) @RT(0) @RT(0)
@END_Attrib
1 0 @F @F @F @F

@Var @RT(7)iDevice @RT(0) @T @F @DT @RT(4)DINT @RT(0) @T @T @BASIC 0 @F
@F @F
@T
@BEG_Attrib
3 @RT(0) @RT(0) @RT(0)
@END_Attrib
1 4 @F @F @F @F

@Var @RT(13)iMoveInDevice @RT(0) @T @F @DT @RT(4)DINT @RT(0) @T @T @BASIC 0 @F
@F @F
@T
@BEG_Attrib
3 @RT(0) @RT(0) @RT(0)
@END_Attrib
1 4 @F @F @F @F

@Var @RT(4)bTmp @RT(0) @T @F @DT @RT(4)BOOL @RT(0) @T @T @BASIC 0 @F
@F @F
@T
@BEG_Attrib
3 @RT(0) @RT(0) @RT(0)
@END_Attrib
1 0 @F @F @F @F

@Var @RT(14)fbSetStepState @RT(0) @T @T @DERIVED 0 @T @T @DT @RT(14)FBSetStepState @RT(0) @T @T @UNKNOWN 0 @F
@F @F
@T
@BEG_Attrib
3 @RT(0) @RT(0) @RT(0)
@END_Attrib
1 0 @F @F @F @F

@Var @RT(1)i @RT(0) @T @F @DT @RT(4)DINT @RT(0) @T @T @BASIC 0 @F
@F @F
@T
@BEG_Attrib
3 @RT(0) @RT(36)movement number at the given StepPos @RT(0)
@END_Attrib
1 4 @F @F @F @F

@Var @RT(5)dummy @RT(0) @T @F @DT @RT(4)DINT @RT(0) @T @T @BASIC 0 @F
@F @F
@T
@BEG_Attrib
3 @RT(0) @RT(0) @RT(0)
@END_Attrib
1 0 @F @F @F @F

@Var @RT(7)bTraced @RT(0) @T @F @DT @RT(4)BOOL @RT(0) @T @T @BASIC 0 @F
@F @F
@T
@BEG_Attrib
3 @RT(0) @RT(0) @RT(0)
@END_Attrib
1 0 @F @F @F @F

@Var @RT(17)iSafetyIdentifier @RT(0) @T @F @DT @RT(4)DINT @RT(0) @T @T @BASIC 0 @F
@F @F
@T
@BEG_Attrib
3 @RT(0) @RT(0) @RT(0)
@END_Attrib
1 0 @F @F @F @F

@Var @RT(8)DeviceId @RT(0) @T @T @DERIVED 0 @T @T @DT @RT(10)tsDeviceId @RT(0) @T @T @UNKNOWN 0 @F
@F @F
@T
@BEG_Attrib
3 @RT(0) @RT(0) @RT(0)
@END_Attrib
1 0 @F @F @F @F

@Var @RT(15)bOverrideSafety @RT(0) @T @F @DT @RT(4)BOOL @RT(0) @T @T @BASIC 0 @F
@F @F
@T
@BEG_Attrib
3 @RT(0) @RT(0) @RT(0)
@END_Attrib
1 0 @F @F @F @F

@Var @RT(9)bDeviceOk @RT(0) @T @F @DT @RT(4)BOOL @RT(0) @T @T @BASIC 0 @F
@F @F
@T
@BEG_Attrib
3 @RT(0) @RT(0) @RT(0)
@END_Attrib
1 0 @F @F @F @F

@Var @RT(15)iValidMovements @RT(0) @T @F @DT @RT(4)DINT @RT(0) @T @T @BASIC 0 @F
@F @F
@T
@BEG_Attrib
3 @RT(0) @RT(0) @RT(0)
@END_Attrib
1 0 @F @F @F @F

@Var @RT(11)iNotOkCount @RT(0) @T @F @DT @RT(4)DINT @RT(0) @T @T @BASIC 0 @F
@F @F
@T
@BEG_Attrib
3 @RT(0) @RT(0) @RT(0)
@END_Attrib
1 3 @F @F @F @F

@END_Dcl

@END_Export

@BEG_Export

@BEG_Algo
@ALGORITHM @RT(6)aCheck @STRUCTURED_TEXT
@RT(0) @RT(0) @RT(0) @F @F
@END_Algo

@BEG_Dcl
@RT(16)DclTreeContainer
5
@Var @RT(7)StepPos @RT(0) @T @T @DERIVED 0 @T @T @DT @RT(12)tsODCStepPos @RT(0) @T @T @UNKNOWN 0 @F
@F @F
@T
@BEG_Attrib
3 @RT(0) @RT(39)Step for which dependencies are checked @RT(0)
@END_Attrib
1 1 @F @F @F @F

@Var @RT(12)DeviceIdSelf @RT(0) @T @T @DERIVED 0 @T @T @DT @RT(10)tsDeviceId @RT(0) @T @T @UNKNOWN 0 @F
@F @F
@T
@BEG_Attrib
3 @RT(0) @RT(31)DeviceId used for error message @RT(0)
@END_Attrib
1 1 @F @F @F @F

@Var @RT(21)bNoAlarmsAndStepState @RT(0) @T @F @DT @RT(4)BOOL @RT(0) @T @T @BASIC 0 @F
@F @F
@T
@BEG_Attrib
3 @RT(0) @RT(65)TRUE: only check dependencies and do not set alarms and stepstate @RT(0)
@END_Attrib
1 1 @F @F @F @F

@Var @RT(8)bAllowed @RT(0) @T @F @DT @RT(4)BOOL @RT(0) @T @T @BASIC 0 @F
@F @F
@T
@BEG_Attrib
3 @RT(0) @RT(26)Dependencies are fulfilled @RT(0)
@END_Attrib
1 3 @F @F @F @F

@Var @RT(11)iNotOkCount @RT(0) @T @F @DT @RT(4)DINT @RT(0) @T @T @BASIC 0 @F
@F @F
@T
@BEG_Attrib
3 @RT(0) @RT(37)number of conditions which are not ok @RT(0)
@END_Attrib
1 3 @F @F @F @F

@END_Dcl

@END_Export

@BEG_Export

@BEG_Algo
@POSTUPDATE_ALGORITHM @RT(22)pOverrideDefaultSafety @STRUCTURED_TEXT
@RT(0) @RT(38)sv_SafetyHMICom.bOverrideDefaultSafety @RT(7)TaskVis @F @F
@END_Algo

@BEG_Dcl
@RT(16)DclTreeContainer
0
@END_Dcl

@END_Export

@BEG_Body
@TL(36)
(**************************************** WARNING ********************************************
 *** The KEBA Kemro K2 System including software is not intended for safety control tasks! ***
 ***                       For further information see Comment tab!                        ***
 *********************************************************************************************)

bAllowed := FALSE;

//find out if it is the first, second, third or fourth instanceable movement in this function unit
iInstanceableMovement := 1;
FOR k := 1 TO cMaxSRInstanceableMovements DO
   IF iMoveInDevice = sv_ODCDeviceMovements.Devices[iDeviceIndex].InstanceableMovements[k] THEN
      iInstanceableMovement := k;
      EXIT;
   END_IF;
END_FOR;

iBegin := cMaxDeviceMovements + ((iInstanceableMovement - 1) * cMaxIntermediateConditions);
tmpDependency := SHL(Dependency, iBegin);

FOR i := 1 TO cMaxIntermediateConditions DO

   tmpDependency := tmpDependency AND cFirstBit;
   IF tmpDependency = cFirstBit THEN
      //bit set => check PosReached of this instance
      bAllowed := sv_ODCDeviceMovements.Devices[iDeviceIndex].Movements[iMoveInDevice]^.InstanceData.pPosReachedArray^[i];

      IF bAllowed THEN
         //movement with posReached = TRUE found -> exit
         EXIT;
      END_IF;
   END_IF;

   tmpDependency := SHL(Dependency, (iBegin + i));

END_FOR;

@END_Body

@@@BEG_Comment@@@
@TL(0)

@@@END_Comment@@@

@BEG_Body
@TL(141)
(**************************************** WARNING ********************************************
 *** The KEBA Kemro K2 System including software is not intended for safety control tasks! ***
 ***                       For further information see Comment tab!                        ***
 *********************************************************************************************)

//check safety array for one step
iNotOkCount := 0;
bAllowed := TRUE;

// when iColumn or iRow = 0 then the movement ist not
// present in the auto cycle (and not safety relevant)
IF StepPos.iColumn = 0 OR StepPos.iRow = 0 THEN
   RETURN;
END_IF;

i := sv_ODCSequenceInt[StepPos.iColumn][StepPos.iRow].iMoveNumber;
IF i = 0 THEN
   //avoid out of range errors
   IF NOT bTraced THEN
      //only trace once and not cyclically
      dummy := Print('!! ABODCCheckDependencies: can not check conditions for movement with move nr. = 0 !!');
      dummy := Print('!! DeviceId: %d/%d  column: %d row: %d !!',DeviceIdSelf.CompId, DeviceIdSelf.IndexId, StepPos.iColumn, StepPos.iRow);
      bTraced := TRUE;
   END_IF;

   bAllowed := FALSE;
   RETURN;
ELSE
   bTraced := FALSE;
END_IF;

iSafetyIdentifier := sv_MovementsAvailable[i].pMovementData^.iSafetyIdentifier;

IF ((NOT mbOverrideDefaultSafety) OR (iSafetyIdentifier = 3)) THEN

   FOR iDevice := 1 TO g_iODCMoveDevicesRegistered DO

      //check override flags
      bOverrideSafety := FALSE;
      DeviceId := sv_ODCDeviceMovements.Devices[iDevice].DeviceId;
      IF ((NOT g_SafetyData.bAvailable) AND sv_bOverrideCoreSafety) AND // override core safety only available if no safetyeditor
         DeviceIdSelf.CompId = cCompCore AND
         (DeviceId.CompId = cCompCore OR DeviceId.CompId = cCompMold OR DeviceId.CompId = cCompEjector) THEN
         (* allow core movements even if mold, other cores or ejector are not in correct position *)
         bOverrideSafety := TRUE;
      END_IF;

      IF ((NOT g_SafetyData.bAvailable) AND sv_bOverrideEjectorSafety) AND // override ejector safety only available if no safetyeditor
         DeviceIdSelf.CompId = cCompEjector AND
         (DeviceId.CompId = cCompCore OR DeviceId.CompId = cCompMold OR DeviceId.CompId = cCompEjector) THEN
         (* allow ejector movements even if mold, cores or possibly other ejectors are not in correct position *)
         bOverrideSafety := TRUE;
      END_IF;

      //check all devices in the safety array
      Dependency := sv_ODCSequenceInt[StepPos.iColumn,StepPos.iRow].SafetyArray[iDevice].Dependency;
      IF (Dependency = cNoDependency) OR bOverrideSafety THEN
         //device is not safety relevant or override is activated
         bDeviceOk := TRUE;
      ELSE
         tmpDependency := Dependency;
         bDeviceOk := FALSE;
         iValidMovements := 0;
         FOR iMoveInDevice := 1 TO sv_ODCDeviceMovements.Devices[iDevice].iNumberOfMovements DO
            //check every movement in this device
            tmpDependency := tmpDependency AND cFirstBit;
            IF tmpDependency = cFirstBit THEN

               iValidMovements := iValidMovements + 1;

               //bit set => check posReached of this movement
               IF sv_ODCDeviceMovements.Devices[iDevice].Movements[iMoveInDevice]^.bInstanceable THEN
                  //instanceable movement => check instances
                  aCheckInstances(Dependency := Dependency,
                                 iDeviceIndex := iDevice,
                                 iMoveInDevice := iMoveInDevice);
                  bTmp := aCheckInstances.bAllowed;
               ELSE
                  bTmp := CHECK_REF(sv_ODCDeviceMovements.Devices[iDevice].Movements[iMoveInDevice]^.pbPosReached^) AND
                              sv_ODCDeviceMovements.Devices[iDevice].Movements[iMoveInDevice]^.pbPosReached^;
               END_IF;

               IF bTmp THEN
                  //valid movement with posReached = TRUE in this device found
                  bDeviceOk := TRUE;
                  EXIT;
               ELSE
                  //continue checking this device and save alarm temporary
                  Alarm := sv_ODCDeviceMovements.Devices[iDevice].Movements[iMoveInDevice]^.Alarm;
               END_IF;
            END_IF;
            tmpDependency := SHL(Dependency, iMoveInDevice);

         END_FOR; //end_for checking all movements in one device

         IF NOT bDeviceOk THEN
            //set correct alarm
            IF NOT bNoAlarmsAndStepState THEN
               IF iValidMovements > 1 THEN
                  //two or more allowed movements: set common alarm erCompNotInCorrectPosition
                  SET_ALARM(Name := erCompNotInCorrectPosition,
                           SubID1 := sv_ODCDeviceMovements.Devices[iDevice].DeviceId.CompId,
                           SubID2 := sv_ODCDeviceMovements.Devices[iDevice].DeviceId.IndexId);
               ELSE
                  //only one valid movement: set alarm of this movement
                  IF (Alarm.AlarmId <> EMPTY) THEN
                     SET_ALARM(Name := Alarm.AlarmId,
                           SubID1 := Alarm.SubId[1],
                           SubID2 := Alarm.SubId[2],
                           SubID3 := Alarm.SubId[3],
                           SubID4 := Alarm.SubId[4],
                           Param1 := Alarm.Param1,
                           Param2 := Alarm.Param2);
                  ELSE
                     SET_ALARM(Name   := erODCComponentLocked,
                                 SubID1 := DeviceIdSelf.CompId,
                                 SubID2 := DeviceIdSelf.IndexId,
                                 SubID3 := sv_ODCDeviceMovements.Devices[iDevice].DeviceId.CompId,
                                 SubID4 := sv_ODCDeviceMovements.Devices[iDevice].DeviceId.IndexId);
                  END_IF;
               END_IF; //end_if iValidMovements
            END_IF;  //end_if bNoAlarmsAndStepState

            //increase counter of not fulfilled conditions
            iNotOkCount := iNotOkCount + 1;

         END_IF; //end_if NOT bDeviceOk

      END_IF; //end_if no dependency or override
      bAllowed := bAllowed AND bDeviceOk;
   END_FOR;  //end_for of checking all devices
END_IF;

IF (iSafetyIdentifier = 1) THEN
   bAllowed := bAllowed AND abSEInterpreter.fCheckMovement(StepPos);
END_IF;

IF (NOT bAllowed) AND (NOT bNoAlarmsAndStepState) THEN
   fbSetStepState(StepPos := StepPos, StepState := nStateError);
END_IF;

@END_Body

@@@BEG_Comment@@@
@TL(1)
check safety array for the given step
@@@END_Comment@@@

@BEG_Body
@TL(9)
(**************************************** WARNING ********************************************
 *** The KEBA Kemro K2 System including software is not intended for safety control tasks! ***
 ***                       For further information see Comment tab!                        ***
 *********************************************************************************************)

aCheckInternal(StepPos := StepPos, DeviceIdSelf := DeviceIdSelf, bNoAlarmsAndStepState := bNoAlarmsAndStepState);
bAllowed := aCheckInternal.bAllowed;
iNotOkCount := aCheckInternal.iNotOkCount;

@END_Body

@@@BEG_Comment@@@
@TL(4)
Check the dependencies of a ODC movement.
Iterates over the dependency array of the step selected by StepPos
and checks the pos reached flags on those movement.
If StepPos.iColumn or StepPos.iRow is 0 then the movement is always allowed.
@@@END_Comment@@@

@BEG_Body
@TL(2)
mbOverrideDefaultSafety := sv_SafetyHMICom.bOverrideDefaultSafety;

@END_Body

@@@BEG_Comment@@@
@TL(0)

@@@END_Comment@@@
@END_Body

@END_Contents
@@@BEG_Password@@@
NGhzZm9kYzQ=
@@@END_Password@@@

(* ---- ABODCDebug.pu ---- *)
(*
@h    ! WARNING !
@h    The Kemro K2 system (including software) only meets category B according to EN 954-1,
@h    thus it is not intended for usage in safety-relevant control applications in the field
@h    of personal safety (e.g. emergency stop).
@h    To implement potentially necessary safety-relevant control tasks, always use additional
@h    external safety devices that are intended for the particular purpose, and meet the necessary
@h    functional safety.
@h    For further information see EN 954-1 (EN ISO 13849-1) and/or the K2-x00 user manual, chapter
@h    "CE conformity, directives and standards".

ODC debug block
- runtime check
- output dependency array to file
*)

IMPORT_OVER_LISTFILE
 ABLogger
, RTC
, tsODCDeviceMovementList
, tyODCSequenceInternal
, tsTraceLevel
, tsODCStepPos
, tyODCDependencyArray
, FBMoveDescription

END_IMPORT

ALGORITHM_BLOCK ABODCDebug #DUMMY_EDIT_BLOCK

SYSTEM_VAR
 sv_ODCDeviceMovements : tsODCDeviceMovementList (* list of all devices that registered movements for the ODC *);
 sv_TraceLevel : tsTraceLevel;
END_VAR

SYSTEM_VAR_IN
 sv_ODCSequenceInt : tyODCSequenceInternal;
END_VAR

VAR_EXTERNAL
 g_iODCMoveDevicesRegistered : DINT;
END_VAR

VAR
 abLogger : ABLogger;
 dStartTime : DATE_AND_TIME;
 dStoppTime : DATE_AND_TIME;
 sTimeDiff : STRING(255);
 dPrint : DINT;
 RealTimeClock : RTC;
 sRunTimeText : STRING(255);
END_VAR

(*
start runtime check, store actual rtc clock
*)

ALGORITHM aRunTimeStart

VAR_INPUT
 sInfoText : STRING(255) := 'undefined instance' (* info for identification of measure object *);
END_VAR
#BEGIN_EDIT_BLOCK
(**************************************** WARNING ********************************************
 *** The KEBA Kemro K2 System including software is not intended for safety control tasks! ***
 ***                       For further information see Comment tab!                        ***
 *********************************************************************************************)

// set info for trace output
sRunTimeText := sInfoText;

// set start time
RealTimeClock(EN := FALSE,
            CDT => dStartTime);

;#END_EDIT_BLOCK END_ALGORITHM

(*
Build difference with start time and output to trace
*)

ALGORITHM aRunTimeStop

#BEGIN_EDIT_BLOCK
(**************************************** WARNING ********************************************
 *** The KEBA Kemro K2 System including software is not intended for safety control tasks! ***
 ***                       For further information see Comment tab!                        ***
 *********************************************************************************************)

// set stop time
RealTimeClock(EN := FALSE,
              CDT => dStoppTime);

// build time difference string
sTimeDiff:= TIME_TO_STRING(SUB_DT_DT(dStoppTime, dStartTime));

IF (sv_TraceLevel.bODCDependencies) THEN
   // write runtime to trace output
   dPrint := Print('%s, runtime = %s', sRunTimeText, sTimeDiff);
END_IF;

;#END_EDIT_BLOCK END_ALGORITHM

ALGORITHM aLogSafety

VAR_INPUT
 sFileName : STRING(255) (* log file name *);
 bAppend : BOOL (* append log file, if false a new file is created and header is written *);
 StepPos : tsODCStepPos (* step position *);
 Dependencies : tyODCDependencyArray (* dependency array to log *);
END_VAR

VAR_TEMP
 i : DINT;
END_VAR

VAR
 sHeadLine1 : STRING(255) (* headline 1 *);
 sHeadLine2 : STRING(255) (* headline 2 *);
 sHeadLine3 : STRING(255) (* headline 3 *);
 sSafetyLine : STRING(255) (* dependency output line *);
 fbMoveDescription : FBMoveDescription;
 sMoveDescription : STRING(255);
END_VAR
#BEGIN_EDIT_BLOCK
(**************************************** WARNING ********************************************
 *** The KEBA Kemro K2 System including software is not intended for safety control tasks! ***
 ***                       For further information see Comment tab!                        ***
 *********************************************************************************************)

IF (NOT bAppend) THEN

   sHeadLine1 := ';';
   sHeadLine2 := ';';
   sHeadLine3 := ';';

   FOR i := 1 TO g_iODCMoveDevicesRegistered BY 1 DO
      sHeadLine1 := CONCAT(sHeadLine1, 'FU_', DINT_TO_STRING(i), ';');
      sHeadLine2 := CONCAT(sHeadLine2, DINT_TO_STRING(sv_ODCDeviceMovements.Devices[i].DeviceId.CompId), '/',
                           DINT_TO_STRING(sv_ODCDeviceMovements.Devices[i].DeviceId.IndexId), ';');
      sHeadLine3 := CONCAT(sHeadLine3, sv_ODCDeviceMovements.Devices[i].sFuName, ';');
   END_FOR;

   abLogger.aWriteLine(sFileName := sFileName,
                        bAppend := FALSE,
                        sText := sHeadLine1);

   abLogger.aWriteLine(sFileName := sFileName,
                        bAppend := TRUE,
                        sText := sHeadLine2);

   abLogger.aWriteLine(sFileName := sFileName,
                        bAppend := TRUE,
                        sText := sHeadLine3);

END_IF;

//get info for this step
fbMoveDescription(iMoveNr := sv_ODCSequenceInt[StepPos.iColumn,StepPos.iRow].iMoveNumber,
                  sDescription => sMoveDescription);

sSafetyLine := CONCAT('Step [', DINT_TO_STRING(StepPos.iColumn),
                      '][', DINT_TO_STRING(StepPos.iRow),
                      ']', ' (', sMoveDescription, ')', ';');

FOR i := 1 TO g_iODCMoveDevicesRegistered BY 1 DO

   IF Dependencies[i].Dependency <> cNoDependency THEN
      sSafetyLine := CONCAT (sSafetyLine, LWORD_TO_STRING(Dependencies[i].Dependency), ';');
   ELSE
      sSafetyLine := CONCAT (sSafetyLine, '-',';');
   END_IF;

   IF (MOD(i, 10) = 0) THEN
      abLogger.aWriteString(sFileName := sFileName,
                            bAppend := TRUE,
                            sText := sSafetyLine);
      sSafetyLine := '';
   END_IF;

END_FOR;

// write rest of string and new line
abLogger.aWriteLine(sFileName := sFileName,
                     bAppend := TRUE,
                     sText := sSafetyLine);

;#END_EDIT_BLOCK END_ALGORITHM

END_ALGORITHM_BLOCK

#END_OF_IEC_PART

@Puma @IecEditor 6 97 @Pou 25
@@@BEG_Comment@@@
@h    ! WARNING !
@h    The Kemro K2 system (including software) only meets category B according to EN 954-1,
@h    thus it is not intended for usage in safety-relevant control applications in the field
@h    of personal safety (e.g. emergency stop).
@h    To implement potentially necessary safety-relevant control tasks, always use additional
@h    external safety devices that are intended for the particular purpose, and meet the necessary
@h    functional safety.
@h    For further information see EN 954-1 (EN ISO 13849-1) and/or the K2-x00 user manual, chapter
@h    "CE conformity, directives and standards".

ODC debug block
- runtime check
- output dependency array to file
@@@END_Comment@@@

@BEG_Contents

@BEG_Func
@RT(17)FuncTreeContainer
0
@END_Func

@BEG_Const
@RT(18)ConstTreeContainer
0
@END_Const

@BEG_Export

@BEG_Kind
@ALGORITHM_BLOCK @RT(10)ABODCDebug @STRUCTURED_TEXT
@RT(0) @RT(0) @RT(0)
@END_Kind

@BEG_Dcl
@RT(16)DclTreeContainer
11
@Var @RT(8)abLogger @RT(0) @T @T @DERIVED 0 @T @T @DT @RT(8)ABLogger @RT(0) @T @T @UNKNOWN 0 @F
@F @F
@T
@BEG_Attrib
3 @RT(0) @RT(0) @RT(0)
@END_Attrib
1 0 @F @F @F @F

@Var @RT(10)dStartTime @RT(0) @T @F @DT @RT(13)DATE_AND_TIME @RT(0) @T @T @BASIC 0 @F
@F @F
@T
@BEG_Attrib
3 @RT(0) @RT(0) @RT(0)
@END_Attrib
1 0 @F @F @F @F

@Var @RT(10)dStoppTime @RT(0) @T @F @DT @RT(13)DATE_AND_TIME @RT(0) @T @T @BASIC 0 @F
@F @F
@T
@BEG_Attrib
3 @RT(0) @RT(0) @RT(0)
@END_Attrib
1 0 @F @F @F @F

@Var @RT(9)sTimeDiff @RT(0) @T @F @DT @RT(11)STRING(255) @RT(0) @T @T @STRING 0 @F @RT(3)255 @F
@F @F
@T
@BEG_Attrib
3 @RT(0) @RT(0) @RT(0)
@END_Attrib
1 0 @F @F @F @F

@Var @RT(6)dPrint @RT(0) @T @F @DT @RT(4)DINT @RT(0) @T @T @BASIC 0 @F
@F @F
@T
@BEG_Attrib
3 @RT(0) @RT(0) @RT(0)
@END_Attrib
1 0 @F @F @F @F

@Var @RT(13)RealTimeClock @RT(0) @T @T @DERIVED 0 @T @T @DT @RT(3)RTC @RT(0) @T @T @UNKNOWN 0 @F
@F @F
@T
@BEG_Attrib
3 @RT(0) @RT(0) @RT(0)
@END_Attrib
1 0 @F @F @F @F

@Var @RT(12)sRunTimeText @RT(0) @T @F @DT @RT(11)STRING(255) @RT(0) @T @T @STRING 0 @F @RT(3)255 @F
@F @F
@T
@BEG_Attrib
3 @RT(0) @RT(0) @RT(0)
@END_Attrib
1 0 @F @F @F @F

@Var @RT(21)sv_ODCDeviceMovements @RT(0) @T @T @DERIVED 0 @T @T @DT @RT(23)tsODCDeviceMovementList @RT(0) @T @T @UNKNOWN 0 @F
@F @F
@T
@BEG_Attrib
3 @RT(0) @RT(57)list of all devices that registered movements for the ODC @RT(0)
@END_Attrib
1 8 @F @F @F @F

@Var @RT(27)g_iODCMoveDevicesRegistered @RT(0) @T @F @DT @RT(4)DINT @RT(0) @T @T @BASIC 0 @F
@F @F
@T
@BEG_Attrib
3 @RT(0) @RT(0) @RT(0)
@END_Attrib
1 6 @F @F @F @F

@Var @RT(17)sv_ODCSequenceInt @RT(0) @T @T @DERIVED 0 @T @T @DT @RT(21)tyODCSequenceInternal @RT(0) @T @T @UNKNOWN 0 @F
@F @F
@T
@BEG_Attrib
3 @RT(0) @RT(0) @RT(0)
@END_Attrib
1 9 @F @F @F @F

@Var @RT(13)sv_TraceLevel @RT(0) @T @T @DERIVED 0 @F @RT(12)tsTraceLevel @F
@T
@BEG_Attrib
3 @RT(0) @RT(0) @RT(0)
@END_Attrib
1 8 @F @F @F @F

@END_Dcl

@END_Export

@BEG_Body

3

@BEG_Export

@BEG_Algo
@ALGORITHM @RT(13)aRunTimeStart @STRUCTURED_TEXT
@RT(0) @RT(0) @RT(0) @F @F
@END_Algo

@BEG_Dcl
@RT(16)DclTreeContainer
1
@Var @RT(9)sInfoText @RT(0) @T @F @DT @RT(11)STRING(255) @RT(0) @T @T @STRING 0 @F @RT(3)255 @F
@F @F
@T
@BEG_Attrib
3 @RT(20)'undefined instance' @RT(41)info for identification of measure object @RT(0)
@END_Attrib
1 1 @F @F @F @F

@END_Dcl

@END_Export

@BEG_Export

@BEG_Algo
@ALGORITHM @RT(12)aRunTimeStop @STRUCTURED_TEXT
@RT(0) @RT(0) @RT(0) @F @F
@END_Algo

@BEG_Dcl
@RT(16)DclTreeContainer
0
@END_Dcl

@END_Export

@BEG_Export

@BEG_Algo
@ALGORITHM @RT(10)aLogSafety @STRUCTURED_TEXT
@RT(0) @RT(0) @RT(0) @F @F
@END_Algo

@BEG_Dcl
@RT(16)DclTreeContainer
11
@Var @RT(9)sFileName @RT(0) @T @F @DT @RT(11)STRING(255) @RT(0) @T @T @STRING 0 @F @RT(3)255 @F
@F @F
@T
@BEG_Attrib
3 @RT(0) @RT(13)log file name @RT(0)
@END_Attrib
1 1 @F @F @F @F

@Var @RT(7)bAppend @RT(0) @T @F @DT @RT(4)BOOL @RT(0) @T @T @BASIC 0 @F
@F @F
@T
@BEG_Attrib
3 @RT(0) @RT(69)append log file, if false a new file is created and header is written @RT(0)
@END_Attrib
1 1 @F @F @F @F

@Var @RT(7)StepPos @RT(0) @T @T @DERIVED 0 @T @T @DT @RT(12)tsODCStepPos @RT(0) @T @T @UNKNOWN 0 @F
@F @F
@T
@BEG_Attrib
3 @RT(0) @RT(13)step position @RT(0)
@END_Attrib
1 1 @F @F @F @F

@Var @RT(12)Dependencies @RT(0) @T @T @DERIVED 0 @F @RT(20)tyODCDependencyArray @F
@T
@BEG_Attrib
3 @RT(0) @RT(23)dependency array to log @RT(0)
@END_Attrib
1 1 @F @F @F @F

@Var @RT(10)sHeadLine1 @RT(0) @T @F @DT @RT(11)STRING(255) @RT(0) @T @T @STRING 0 @F @RT(3)255 @F
@F @F
@T
@BEG_Attrib
3 @RT(0) @RT(10)headline 1 @RT(0)
@END_Attrib
1 0 @F @F @F @F

@Var @RT(10)sHeadLine2 @RT(0) @T @F @DT @RT(11)STRING(255) @RT(0) @T @T @STRING 0 @F @RT(3)255 @F
@F @F
@T
@BEG_Attrib
3 @RT(0) @RT(10)headline 2 @RT(0)
@END_Attrib
1 0 @F @F @F @F

@Var @RT(10)sHeadLine3 @RT(0) @T @F @DT @RT(11)STRING(255) @RT(0) @T @T @STRING 0 @F @RT(3)255 @F
@F @F
@T
@BEG_Attrib
3 @RT(0) @RT(10)headline 3 @RT(0)
@END_Attrib
1 0 @F @F @F @F

@Var @RT(11)sSafetyLine @RT(0) @T @F @DT @RT(11)STRING(255) @RT(0) @T @T @STRING 0 @F @RT(3)255 @F
@F @F
@T
@BEG_Attrib
3 @RT(0) @RT(22)dependency output line @RT(0)
@END_Attrib
1 0 @F @F @F @F

@Var @RT(1)i @RT(0) @T @F @DT @RT(4)DINT @RT(0) @T @T @BASIC 0 @F
@F @F
@T
@BEG_Attrib
3 @RT(0) @RT(0) @RT(0)
@END_Attrib
1 4 @F @F @F @F

@Var @RT(17)fbMoveDescription @RT(0) @T @T @DERIVED 0 @T @T @DT @RT(17)FBMoveDescription @RT(0) @T @T @UNKNOWN 0 @F
@F @F
@T
@BEG_Attrib
3 @RT(0) @RT(0) @RT(0)
@END_Attrib
1 0 @F @F @F @F

@Var @RT(16)sMoveDescription @RT(0) @T @F @DT @RT(11)STRING(255) @RT(0) @T @T @STRING 0 @F @RT(3)255 @F
@F @F
@T
@BEG_Attrib
3 @RT(0) @RT(0) @RT(0)
@END_Attrib
1 0 @F @F @F @F

@END_Dcl

@END_Export

@BEG_Body
@TL(12)
(**************************************** WARNING ********************************************
 *** The KEBA Kemro K2 System including software is not intended for safety control tasks! ***
 ***                       For further information see Comment tab!                        ***
 *********************************************************************************************)

// set info for trace output
sRunTimeText := sInfoText;

// set start time
RealTimeClock(EN := FALSE,
            CDT => dStartTime);

@END_Body

@@@BEG_Comment@@@
@TL(1)
start runtime check, store actual rtc clock
@@@END_Comment@@@

@BEG_Body
@TL(18)
(**************************************** WARNING ********************************************
 *** The KEBA Kemro K2 System including software is not intended for safety control tasks! ***
 ***                       For further information see Comment tab!                        ***
 *********************************************************************************************)

// set stop time
RealTimeClock(EN := FALSE,
              CDT => dStoppTime);

// build time difference string
sTimeDiff:= TIME_TO_STRING(SUB_DT_DT(dStoppTime, dStartTime));

IF (sv_TraceLevel.bODCDependencies) THEN
   // write runtime to trace output
   dPrint := Print('%s, runtime = %s', sRunTimeText, sTimeDiff);
END_IF;

@END_Body

@@@BEG_Comment@@@
@TL(1)
Build difference with start time and output to trace
@@@END_Comment@@@

@BEG_Body
@TL(63)
(**************************************** WARNING ********************************************
 *** The KEBA Kemro K2 System including software is not intended for safety control tasks! ***
 ***                       For further information see Comment tab!                        ***
 *********************************************************************************************)

IF (NOT bAppend) THEN

   sHeadLine1 := ';';
   sHeadLine2 := ';';
   sHeadLine3 := ';';

   FOR i := 1 TO g_iODCMoveDevicesRegistered BY 1 DO
      sHeadLine1 := CONCAT(sHeadLine1, 'FU_', DINT_TO_STRING(i), ';');
      sHeadLine2 := CONCAT(sHeadLine2, DINT_TO_STRING(sv_ODCDeviceMovements.Devices[i].DeviceId.CompId), '/',
                           DINT_TO_STRING(sv_ODCDeviceMovements.Devices[i].DeviceId.IndexId), ';');
      sHeadLine3 := CONCAT(sHeadLine3, sv_ODCDeviceMovements.Devices[i].sFuName, ';');
   END_FOR;

   abLogger.aWriteLine(sFileName := sFileName,
                        bAppend := FALSE,
                        sText := sHeadLine1);

   abLogger.aWriteLine(sFileName := sFileName,
                        bAppend := TRUE,
                        sText := sHeadLine2);

   abLogger.aWriteLine(sFileName := sFileName,
                        bAppend := TRUE,
                        sText := sHeadLine3);

END_IF;

//get info for this step
fbMoveDescription(iMoveNr := sv_ODCSequenceInt[StepPos.iColumn,StepPos.iRow].iMoveNumber,
                  sDescription => sMoveDescription);

sSafetyLine := CONCAT('Step [', DINT_TO_STRING(StepPos.iColumn),
                      '][', DINT_TO_STRING(StepPos.iRow),
                      ']', ' (', sMoveDescription, ')', ';');

FOR i := 1 TO g_iODCMoveDevicesRegistered BY 1 DO

   IF Dependencies[i].Dependency <> cNoDependency THEN
      sSafetyLine := CONCAT (sSafetyLine, LWORD_TO_STRING(Dependencies[i].Dependency), ';');
   ELSE
      sSafetyLine := CONCAT (sSafetyLine, '-',';');
   END_IF;

   IF (MOD(i, 10) = 0) THEN
      abLogger.aWriteString(sFileName := sFileName,
                            bAppend := TRUE,
                            sText := sSafetyLine);
      sSafetyLine := '';
   END_IF;

END_FOR;

// write rest of string and new line
abLogger.aWriteLine(sFileName := sFileName,
                     bAppend := TRUE,
                     sText := sSafetyLine);

@END_Body

@@@BEG_Comment@@@
@TL(0)

@@@END_Comment@@@
@END_Body

@END_Contents
@@@BEG_Password@@@
NGhzZm9kYzQ=
@@@END_Password@@@
